{attribute 'GeneratedUsingTerminal: CU2508-0000-0017'}
{attribute addProperty BoxType "CU2508-0000-0017"}
{attribute addProperty Id "Dropped_frames_rxAT %I*USINT1Dropped_frames_txAT %I*USINT1"}
{attribute addProperty CRC "945715530"}
{attribute addProperty Size "2"}
TYPE EPM_Inputs_Channel_385E794A EXTENDS InputBase_8311D824 :
STRUCT
	{attribute addProperty Name "Dropped_frames_rx"}
	Dropped_frames_rx AT %I* : USINT;
	{attribute addProperty Name "Dropped_frames_tx"}
	Dropped_frames_tx AT %I* : USINT;
END_STRUCT
END_TYPE

(* stored: Version 1.2.0.0, ProductVersion 3.1.4024.9
   DUT EPM_Inputs_Channel_385E794A: Id {071f6e22-1178-4be2-94cf-c171c8aca3bc} *)
